// TIA Portal project "3M series" (V16)

(* hardware
DEVICE "S7-1200 station_1"  S7-1200 Station
   slot 0: "Rack_0"  S7-1200 Rack  Rack  V1.0
   slot 1: "PLC_1"  CPU 1212C AC/DC/Rly  6ES7 212-1BE40-0XB0  V4.0
*)

// ===== PLC "PLC_1"  CPU 1212C AC/DC/Rly =====

VAR_GLOBAL   // PLC tag table "Default tag table"
   "stop" AT %I0.0 : Bool;
   "start" AT %I0.1 : Bool;
   "motor 1" AT %Q0.0 : Bool;
   "motor 2" AT %Q0.1 : Bool;
   "motor 3" AT %Q0.2 : Bool;
   "Loop Marker" AT %M0.0 : Bool;
   "M1 ss" AT %M0.1 : Bool;
   "M2 ss" AT %M0.2 : Bool;
   "M3 ss" AT %M0.3 : Bool;
   "M2 series" AT %M0.4 : Bool;
END_VAR

// folder: System blocks/Program resources

DATA_BLOCK "T1"   // DB1
{ S7_Optimized_Access := 'TRUE' }
AUTHOR : Simatic
FAMILY : IEC
NAME : IEC_TMR
VERSION : 1.0
// stored: InstanceOfName IEC_TIMER
"IEC_TIMER"
BEGIN
END_DATA_BLOCK

DATA_BLOCK "T2"   // DB2
{ S7_Optimized_Access := 'TRUE' }
AUTHOR : Simatic
FAMILY : IEC
NAME : IEC_TMR
VERSION : 1.0
// stored: InstanceOfName IEC_TIMER
"IEC_TIMER"
BEGIN
END_DATA_BLOCK

DATA_BLOCK "T3"   // DB3
{ S7_Optimized_Access := 'TRUE' }
AUTHOR : Simatic
FAMILY : IEC
NAME : IEC_TMR
VERSION : 1.0
// stored: InstanceOfName IEC_TIMER
"IEC_TIMER"
BEGIN
END_DATA_BLOCK

DATA_BLOCK "T4"   // DB4
{ S7_Optimized_Access := 'TRUE' }
AUTHOR : Simatic
FAMILY : IEC
NAME : IEC_TMR
VERSION : 1.0
// stored: InstanceOfName IEC_TIMER
"IEC_TIMER"
BEGIN
END_DATA_BLOCK

// folder: (top level)

ORGANIZATION_BLOCK "Main"   // OB1, LAD, ProgramCycle
TITLE = "Main Program Sweep (Cycle)"
{ S7_Optimized_Access := 'TRUE' }
VERSION : 0.1
   VAR_INPUT
      Initial_Call : Bool;   // Initial call of this OB
      Remanence : Bool;   // =True, if remanent data are available
   END_VAR
BEGIN

REGION Network 1
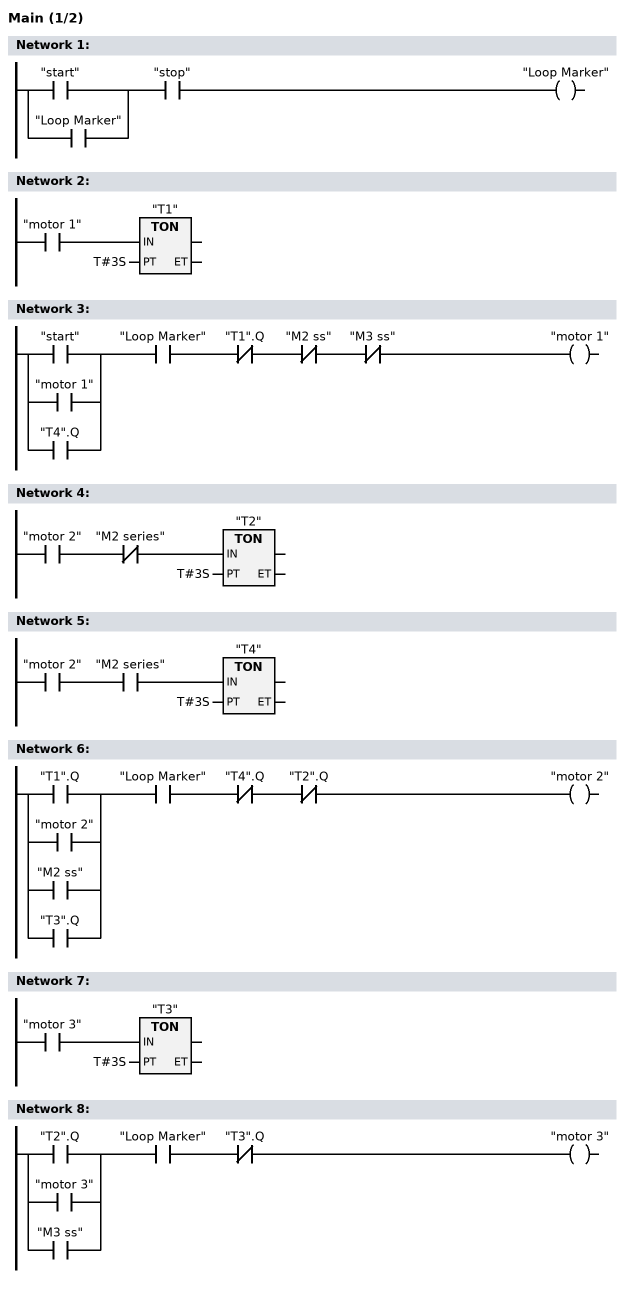
   RUNG wire#powerrail
      Contact( "start" )
      wire#w1
      Contact( "stop" )
      Coil( "Loop Marker" )
   END_RUNG
   RUNG wire#powerrail
      Contact( "Loop Marker" )
   END_RUNG wire#w1
   // the same network as SCL:
   "Loop Marker" := ("start" OR "Loop Marker") AND "stop";
END_REGION

REGION Network 2
   "T1".TON(IN := "motor 1", PT := T#3S);
END_REGION

REGION Network 3
   RUNG wire#powerrail
      Contact( "start" )
      wire#w1
      Contact( "Loop Marker" )
      I_Contact( "T1".Q )
      I_Contact( "M2 ss" )
      I_Contact( "M3 ss" )
      Coil( "motor 1" )
   END_RUNG
   RUNG wire#powerrail
      Contact( "motor 1" )
   END_RUNG wire#w1
   RUNG wire#powerrail
      Contact( "T4".Q )
   END_RUNG wire#w1
   // the same network as SCL:
   "motor 1" := ("start" OR "motor 1" OR "T4".Q) AND "Loop Marker" AND NOT "T1".Q AND NOT "M2 ss" AND NOT "M3 ss";
END_REGION

REGION Network 4
   "T2".TON(IN := "motor 2" AND NOT "M2 series", PT := T#3S);
END_REGION

REGION Network 5
   "T4".TON(IN := "motor 2" AND "M2 series", PT := T#3S);
END_REGION

REGION Network 6
   RUNG wire#powerrail
      Contact( "T1".Q )
      wire#w1
      Contact( "Loop Marker" )
      I_Contact( "T4".Q )
      I_Contact( "T2".Q )
      Coil( "motor 2" )
   END_RUNG
   RUNG wire#powerrail
      Contact( "motor 2" )
   END_RUNG wire#w1
   RUNG wire#powerrail
      Contact( "M2 ss" )
   END_RUNG wire#w1
   RUNG wire#powerrail
      Contact( "T3".Q )
   END_RUNG wire#w1
   // the same network as SCL:
   "motor 2" := ("T1".Q OR "motor 2" OR "M2 ss" OR "T3".Q) AND "Loop Marker" AND NOT "T4".Q AND NOT "T2".Q;
END_REGION

REGION Network 7
   "T3".TON(IN := "motor 3", PT := T#3S);
END_REGION

REGION Network 8
   RUNG wire#powerrail
      Contact( "T2".Q )
      wire#w1
      Contact( "Loop Marker" )
      I_Contact( "T3".Q )
      Coil( "motor 3" )
   END_RUNG
   RUNG wire#powerrail
      Contact( "motor 3" )
   END_RUNG wire#w1
   RUNG wire#powerrail
      Contact( "M3 ss" )
   END_RUNG wire#w1
   // the same network as SCL:
   "motor 3" := ("T2".Q OR "motor 3" OR "M3 ss") AND "Loop Marker" AND NOT "T3".Q;
END_REGION

REGION Network 9
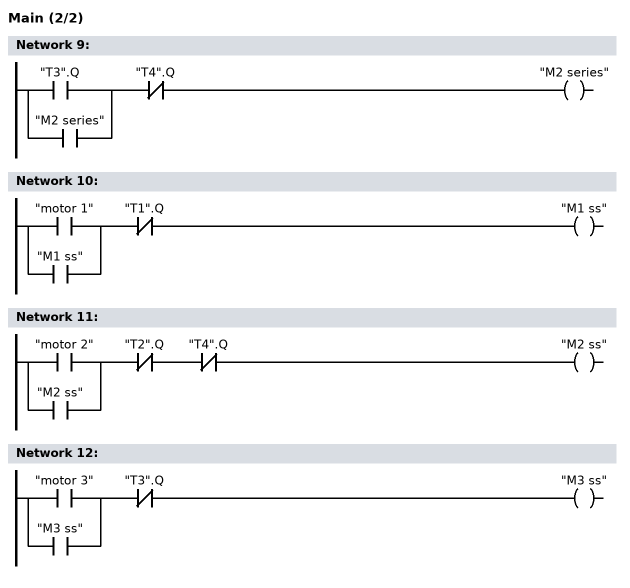
   RUNG wire#powerrail
      Contact( "T3".Q )
      wire#w1
      I_Contact( "T4".Q )
      Coil( "M2 series" )
   END_RUNG
   RUNG wire#powerrail
      Contact( "M2 series" )
   END_RUNG wire#w1
   // the same network as SCL:
   "M2 series" := ("T3".Q OR "M2 series") AND NOT "T4".Q;
END_REGION

REGION Network 10
   RUNG wire#powerrail
      Contact( "motor 1" )
      wire#w1
      I_Contact( "T1".Q )
      Coil( "M1 ss" )
   END_RUNG
   RUNG wire#powerrail
      Contact( "M1 ss" )
   END_RUNG wire#w1
   // the same network as SCL:
   "M1 ss" := ("motor 1" OR "M1 ss") AND NOT "T1".Q;
END_REGION

REGION Network 11
   RUNG wire#powerrail
      Contact( "motor 2" )
      wire#w1
      I_Contact( "T2".Q )
      I_Contact( "T4".Q )
      Coil( "M2 ss" )
   END_RUNG
   RUNG wire#powerrail
      Contact( "M2 ss" )
   END_RUNG wire#w1
   // the same network as SCL:
   "M2 ss" := ("motor 2" OR "M2 ss") AND NOT "T2".Q AND NOT "T4".Q;
END_REGION

REGION Network 12
   RUNG wire#powerrail
      Contact( "motor 3" )
      wire#w1
      I_Contact( "T3".Q )
      Coil( "M3 ss" )
   END_RUNG
   RUNG wire#powerrail
      Contact( "M3 ss" )
   END_RUNG wire#w1
   // the same network as SCL:
   "M3 ss" := ("motor 3" OR "M3 ss") AND NOT "T3".Q;
END_REGION
END_ORGANIZATION_BLOCK